// This function has been automatically generated from the project information.
{attribute 'signature_flag' := '1073741824'}
{attribute 'TcGenerated'}
{attribute 'no-analysis'}
FUNCTION F_GetCompany : WSTRING
VAR_INPUT
	
END_VAR

F_GetCompany := "AU-tomation";

END_FUNCTION

(* stored: Version 1.1.0.1
   POU F_GetCompany: Id {4fb1a900-3564-4f40-9de4-2fc1f57ed872}, SpecialFunc None *)
